// TIA Portal project "P11_2" (V20)

(* hardware
DEVICE "HMI_1"  KTP700 Basic PN
   slot 0: "HMI_1"  KTP700 Basic PN  6AV2 123-2GB03-0AX0  17.0.0.0
   slot 1: "HMI_RT_1"  KTP700 Basic PN  6AV2 123-2GB03-0AX0  17.0.0.0
   slot 5: "HMI_1.IE_CP_1"  PROFINET Interface  17.0.0.0
      slot 1: "PROFINET Interface_1"  PROFINET Interface
         slot 1: "Port_1"  Port
DEVICE "S7-1200 station_1"  S7-1200 Station
   slot 0: "Rack_0"  S7-1200 Rack  Rack  V1.0
   slot 1: "PLC_1"  CPU 1214C DC/DC/DC  6ES7 214-1AG40-0XB0  V4.7
*)

// ===== PLC "PLC_1"  CPU 1214C DC/DC/DC =====

VAR_GLOBAL   // PLC tag table "Default tag table"
   "Inicio" AT %M0.2 : Bool;
   "Marca 1" AT %M0.1 : Bool;
   "Marca0" AT %M0.0 : Bool;
   "Reset" AT %M0.4 : Bool;
   "SalidaControl" AT %M0.3 : Bool;
   "Tiempo_out_ms" AT %MD200 : Time;
   "Tiempo_out_seg" AT %MD66 : Real;
   "Tiempo_in" AT %MD150 : DInt;
   "Tiempo_in_ms" AT %MD184 : DInt;
   "Salida led" AT %M0.5 : Bool;
   "Regla3_1" AT %M26.0 : LReal;
   "Salida_barra" AT %M34.0 : LReal;
   "Tag_1" AT %Q0.0 : Bool;
   "Verde" AT %M2.0 : Bool;
   "Amarillo" AT %M2.1 : Bool;
   "Rojo" AT %M2.2 : Bool;
   "reset_rojo" AT %M2.3 : Bool;
   "reset_sem" AT %M2.4 : Bool;
   "cont_verde" AT %MD100 : Time;
   "cont_ama" AT %MD104 : Time;
   "cont_rojo" AT %MD108 : Time;
   "Tag_2" AT %MD12 : DInt;
   "T_restante" AT %MD16 : DInt;
   "Tag_3" AT %MD20 : DInt;
   "Tag_4" AT %MD24 : DInt;
   "Tag_5" AT %M26.0 : Bool;
   "Alarma1" AT %MW42 : Word;
   "bitalarma1" AT %M43.0 : Bool;
   "Alarma2" AT %MW44 : Word;
   "bitAlarma2" AT %M45.0 : Bool;
   "Alarma3" AT %MW46 : Word;
   "bitalarma3" AT %M47.0 : Bool;
END_VAR

// folder: System blocks/Program resources

DATA_BLOCK "IEC_Timer_0_DB"   // DB1
{ S7_Optimized_Access := 'TRUE' }
AUTHOR : Simatic
FAMILY : IEC
NAME : IEC_TMR
VERSION : 1.0
// stored: InstanceOfName IEC_TIMER
"IEC_TIMER"
BEGIN
END_DATA_BLOCK

DATA_BLOCK "IEC_Timer_0_DB_1"   // DB2
{ S7_Optimized_Access := 'TRUE' }
AUTHOR : Simatic
FAMILY : IEC
NAME : IEC_TMR
VERSION : 1.0
// stored: InstanceOfName IEC_TIMER
"IEC_TIMER"
BEGIN
END_DATA_BLOCK

DATA_BLOCK "IEC_Timer_0_DB_2"   // DB3
{ S7_Optimized_Access := 'TRUE' }
AUTHOR : Simatic
FAMILY : IEC
NAME : IEC_TMR
VERSION : 1.0
// stored: InstanceOfName IEC_TIMER
"IEC_TIMER"
BEGIN
END_DATA_BLOCK

DATA_BLOCK "IEC_Timer_0_DB_3"   // DB4
{ S7_Optimized_Access := 'TRUE' }
AUTHOR : Simatic
FAMILY : IEC
NAME : IEC_TMR
VERSION : 1.0
// stored: InstanceOfName IEC_TIMER
"IEC_TIMER"
BEGIN
END_DATA_BLOCK

// folder: (top level)

ORGANIZATION_BLOCK "Main"   // OB1, LAD, ProgramCycle
TITLE = "Main Program Sweep (Cycle)"
{ S7_Optimized_Access := 'TRUE' }
VERSION : 0.1
   VAR_INPUT
      Initial_Call : Bool;   // Initial call of this OB
      Remanence : Bool;   // =True, if remanent data are available
   END_VAR
BEGIN

REGION Network 1
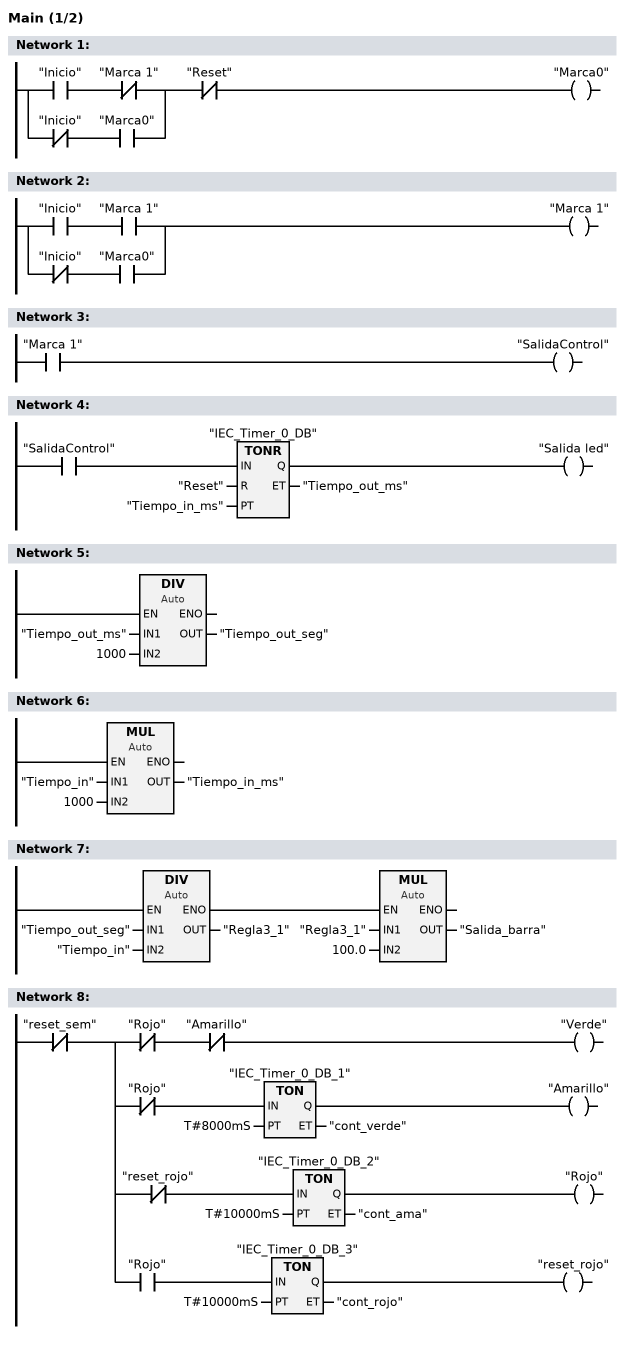
   RUNG wire#powerrail
      Contact( "Inicio" )
      I_Contact( "Marca 1" )
      wire#w1
      I_Contact( "Reset" )
      Coil( "Marca0" )
   END_RUNG
   RUNG wire#powerrail
      I_Contact( "Inicio" )
      Contact( "Marca0" )
   END_RUNG wire#w1
   // the same network as SCL:
   "Marca0" := (("Inicio" AND NOT "Marca 1") OR (NOT "Inicio" AND "Marca0")) AND NOT "Reset";
END_REGION

REGION Network 2
   RUNG wire#powerrail
      Contact( "Inicio" )
      Contact( "Marca 1" )
      wire#w1
      Coil( "Marca 1" )
   END_RUNG
   RUNG wire#powerrail
      I_Contact( "Inicio" )
      Contact( "Marca0" )
   END_RUNG wire#w1
   // the same network as SCL:
   "Marca 1" := ("Inicio" AND "Marca 1") OR (NOT "Inicio" AND "Marca0");
END_REGION

REGION Network 3
   RUNG wire#powerrail
      Contact( "Marca 1" )
      Coil( "SalidaControl" )
   END_RUNG
   // the same network as SCL:
   "SalidaControl" := "Marca 1";
END_REGION

REGION Network 4
   "IEC_Timer_0_DB".TONR(IN := "SalidaControl", R := "Reset", PT := "Tiempo_in_ms", ET => "Tiempo_out_ms");
   "Salida led" := "IEC_Timer_0_DB".Q;
END_REGION

REGION Network 5
   RUNG wire#powerrail
      Div(in1 := "Tiempo_out_ms", in2 := 1000, out => "Tiempo_out_seg")
   END_RUNG
   // the same network as SCL:
   "Tiempo_out_seg" := "Tiempo_out_ms" / 1000;
END_REGION

REGION Network 6
   RUNG wire#powerrail
      Mul(in1 := "Tiempo_in", in2 := 1000, out => "Tiempo_in_ms")
   END_RUNG
   // the same network as SCL:
   "Tiempo_in_ms" := "Tiempo_in" * 1000;
END_REGION

REGION Network 7
   RUNG wire#powerrail
      Div(in1 := "Tiempo_out_seg", in2 := "Tiempo_in", out => "Regla3_1")
      Mul(in1 := "Regla3_1", in2 := 100.0, out => "Salida_barra")
   END_RUNG
   // the same network as SCL:
   "Regla3_1" := "Tiempo_out_seg" / "Tiempo_in";
   "Salida_barra" := "Regla3_1" * 100.0;
END_REGION

REGION Network 8
   "Verde" := NOT "reset_sem" AND NOT "Rojo" AND NOT "Amarillo";
   "IEC_Timer_0_DB_1".TON(IN := NOT "reset_sem" AND NOT "Rojo", PT := T#8000mS, ET => "cont_verde");
   "Amarillo" := "IEC_Timer_0_DB_1".Q;
   "IEC_Timer_0_DB_2".TON(IN := NOT "reset_sem" AND NOT "reset_rojo", PT := T#10000mS, ET => "cont_ama");
   "Rojo" := "IEC_Timer_0_DB_2".Q;
   "IEC_Timer_0_DB_3".TON(IN := NOT "reset_sem" AND "Rojo", PT := T#10000mS, ET => "cont_rojo");
   "reset_rojo" := "IEC_Timer_0_DB_3".Q;
END_REGION

REGION Network 9
   // T restante verde
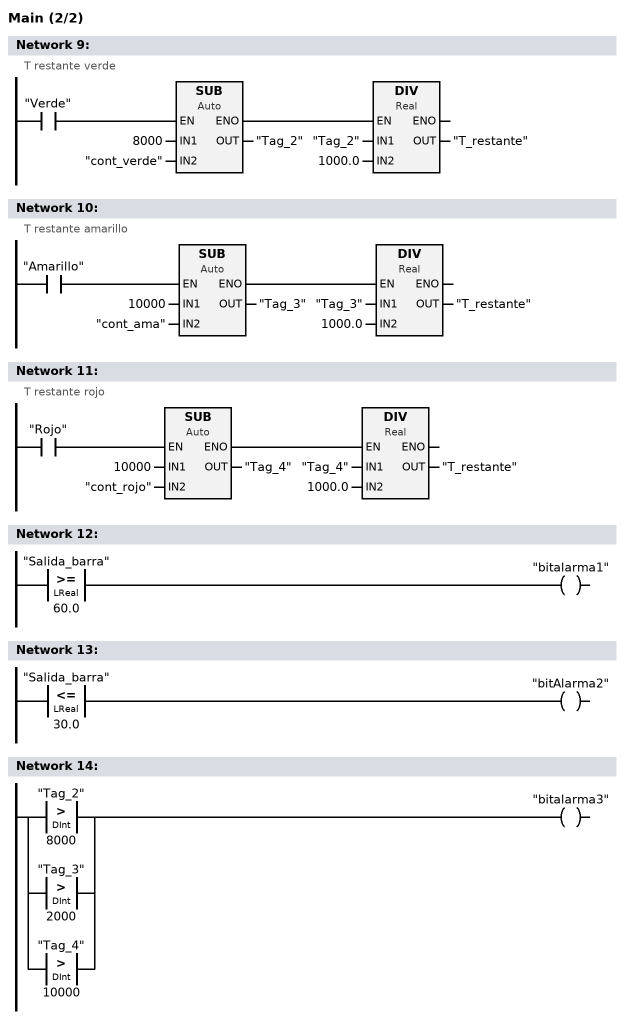
   RUNG wire#powerrail
      Contact( "Verde" )
      Sub(in1 := 8000, in2 := "cont_verde", out => "Tag_2")
      { S7_Templates := "SrcType := Real" } Div(in1 := "Tag_2", in2 := 1000.0, out => "T_restante")
   END_RUNG
   // the same network as SCL:
   IF "Verde" THEN
       "Tag_2" := 8000 - "cont_verde";
       "T_restante" := "Tag_2" / 1000.0;
   END_IF;
END_REGION

REGION Network 10
   // T restante amarillo
   RUNG wire#powerrail
      Contact( "Amarillo" )
      Sub(in1 := 10000, in2 := "cont_ama", out => "Tag_3")
      { S7_Templates := "SrcType := Real" } Div(in1 := "Tag_3", in2 := 1000.0, out => "T_restante")
   END_RUNG
   // the same network as SCL:
   IF "Amarillo" THEN
       "Tag_3" := 10000 - "cont_ama";
       "T_restante" := "Tag_3" / 1000.0;
   END_IF;
END_REGION

REGION Network 11
   // T restante rojo
   RUNG wire#powerrail
      Contact( "Rojo" )
      Sub(in1 := 10000, in2 := "cont_rojo", out => "Tag_4")
      { S7_Templates := "SrcType := Real" } Div(in1 := "Tag_4", in2 := 1000.0, out => "T_restante")
   END_RUNG
   // the same network as SCL:
   IF "Rojo" THEN
       "Tag_4" := 10000 - "cont_rojo";
       "T_restante" := "Tag_4" / 1000.0;
   END_IF;
END_REGION

REGION Network 12
   RUNG wire#powerrail
      { S7_Templates := "SrcType := LReal" } GE_Contact(in1 := "Salida_barra", in2 := 60.0)
      Coil( "bitalarma1" )
   END_RUNG
   // the same network as SCL:
   "bitalarma1" := "Salida_barra" >= 60.0;
END_REGION

REGION Network 13
   RUNG wire#powerrail
      { S7_Templates := "SrcType := LReal" } LE_Contact(in1 := "Salida_barra", in2 := 30.0)
      Coil( "bitAlarma2" )
   END_RUNG
   // the same network as SCL:
   "bitAlarma2" := "Salida_barra" <= 30.0;
END_REGION

REGION Network 14
   RUNG wire#powerrail
      { S7_Templates := "SrcType := DInt" } GT_Contact(in1 := "Tag_2", in2 := 8000)
      wire#w1
      Coil( "bitalarma3" )
   END_RUNG
   RUNG wire#powerrail
      { S7_Templates := "SrcType := DInt" } GT_Contact(in1 := "Tag_3", in2 := 2000)
   END_RUNG wire#w1
   RUNG wire#powerrail
      { S7_Templates := "SrcType := DInt" } GT_Contact(in1 := "Tag_4", in2 := 10000)
   END_RUNG wire#w1
   // the same network as SCL:
   "bitalarma3" := ("Tag_2" > 8000) OR ("Tag_3" > 2000) OR ("Tag_4" > 10000);
END_REGION
END_ORGANIZATION_BLOCK

(* ===== HMI "HMI_RT_1" =====
system functions are stored by id; their names below are inferred from use
connection "HMI_Connection_1": ETHERNET, SMART_S7_1200_OMS

HMI tags "Default tag table"
   "Tag_ScreenNumber" : UInt, internal
   "Inicio" : Bool = PLC Inicio AT %M0.2, 1 s
   "Reset" : Bool = PLC Reset AT %M0.4, 1 s
   "Tiempo_in" : DInt = PLC Tiempo_in AT %MD150, 1 s
   "Tiempo_out_seg" : Real = PLC Tiempo_out_seg AT %MD66, 1 s
   "Salida_barra" : LReal = PLC Salida_barra AT %M34.0, 1 s
   "Salida led" : Bool = PLC "Salida led" AT %M0.5, 1 s
   "Rojo" : Bool = PLC Rojo AT %M2.2, 1 s
   "Amarillo" : Bool = PLC Amarillo AT %M2.1, 1 s
   "Verde" : Bool = PLC Verde AT %M2.0, 1 s
   "T_restante" : DInt = PLC T_restante AT %MD16, 1 s
   "reset_sem" : Bool = PLC reset_sem AT %M2.4, 1 s
   "Alarma1" : Word = PLC Alarma1 AT %MW42, 1 s
   "Alarma2" : Word = PLC Alarma2 AT %MW44, 1 s
   "Alarma3" : Word = PLC Alarma3 AT %MW46, 1 s

discrete alarms
   1: 'Ha sobrepasado el 60%', class Errors, trigger "Alarma1" bit 0
   2: 'El nivel es menor al 30%', class Warnings, trigger "Alarma2" bit 0
   3: 'Tiempo establecido para cada estado no cumplido', class Acknowledgement, trigger "Alarma3" bit 0

text list "list_verde": 1 'AVANCE'; 0 ''

text list "list_rojo": 1 '¡ALTO!'; 0 ''

text list "list_ama": 1 'PRECAUCIÓN'; 0 ''

Template "Template_1" 800x480
   Button "Exit" at 714,429 size 71x50; TextOff 'Exit'; PictureOff "ExitRuntime_KTP700_Basic_PN_TR"; PictureOn "ExitRuntime_KTP700_Basic_PN_TR"
      on Release: StopRuntime(0)
   Button "Template_Button" at 614,429 size 71x50; TextOff 'Text'
   Button "Template_Button_1" at 514,429 size 71x50; TextOff 'Text'
   Button "Template_Button_2" at 414,429 size 71x50; TextOff 'Text'
   Button "Template_Button_3" at 314,429 size 71x50; TextOff 'Text'
   Button "Template_Button_4" at 214,429 size 71x50; TextOff 'Text'
   Button "Template_Button_5" at 114,429 size 71x50; TextOff 'Text'
   Button "Start screen" at 14,429 size 71x50; TextOff 'Start screen'; PictureOff "NavigateHome_KTP700_Basic_PN_TR"; PictureOn "NavigateHome_KTP700_Basic_PN_TR"
      on Release: ActivateScreen("Root screen", 0)
   SymbolicIOField "Symbolic_IO_Field_Screen" at 93,9 size 600x33; TextOff '0'; TextOn '1'; TextList "TextList_ScreenNames"
      ProcessValue <- "Tag_ScreenNumber"
      on Change: ActivateScreenByNumber("Tag_ScreenNumber", 0)
   DateTimeField "HmiScreenItemData" at 695,25 size 105x25
   DateTimeField "HmiScreenItemData_1" at 695,0 size 105x25
   GraphicView "Logo" at 0,0 size 91x51; Picture "Logo of HMI_1"

screen "Root screen" 800x480, template "Template_1"
   on GenerateScreen: SetTag("Tag_ScreenNumber", 1)
   Button "Button_1" at 633,377 size 145x32; TextOff 'Reset'
      on Press: SetBit("reset_sem")
      on Release: ResetBit("reset_sem")
   IOField "I/O field_1" at 455,160 size 79x39; FormatPattern 99; Unit s
      ProcessValue <- "T_restante"
   TextField "Text field_1" at 423,132 size 140x23; Text 'Tiempo restante'
   Circle "Circle_1" at 285,124 size 48x48
      Appearance <- "Rojo"
   Circle "Circle_2" at 284,199 size 48x48
      Appearance <- "Amarillo"
   Circle "Circle_3" at 283,267 size 48x48
      Appearance <- "Verde"
   SymbolicIOField "Symbolic I/O field_1" at 426,299 size 137x32; TextOff '0'; TextOn '1'; TextList "list_verde"
      ProcessValue <- "Verde"
   SymbolicIOField "Symbolic I/O field_2" at 426,264 size 136x32; TextOff '0'; TextOn '1'; TextList "list_ama"
      ProcessValue <- "Amarillo"
   SymbolicIOField "Symbolic I/O field_3" at 426,229 size 135x32; TextOff '0'; TextOn '1'; TextList "list_rojo"
      ProcessValue <- "Rojo"
   Button "FB_ArrowRight_Square" at 36,60 size 50x50; TextOff 'Text'; PictureOff "FB_ArrowRight_Square_Released_256c"; PictureOn "FB_ArrowRight_Square_Pressed_256c"
      on Press: ActivateScreen("tanque", 0)

screen "tanque" 800x480
   Bar "Bar_1" at 113,70 size 92x283; MinimumValue 0; MaximumValue 100
      ProcessValue <- "Salida_barra"
   TextField "Text field_1" at 249,149 size 143x23; Text 'Límite de tiempo'
   TextField "Text field_2" at 477,148 size 174x23; Text 'Tiempo Transcurrido'
   Button "Button_1" at 266,246 size 126x32; TextOff 'Inicio/Pausa'
      on Press: SetBit("Inicio")
      on Release: ResetBit("Inicio")
   Button "Button_2" at 477,246 size 128x32; TextOff 'Reset'
      on Press: SetBit("Reset")
      on Release: ResetBit("Reset")
   IOField "I/O field_1" at 267,177 size 96x32; FormatPattern 999; Unit  seg
      ProcessValue <- "Tiempo_in"
   IOField "I/O field_2" at 509,178 size 96x32; FormatPattern 999; Unit  seg
      ProcessValue <- "Tiempo_out_seg"
   Circle "Circle_1" at 416,246 size 34x34
      Appearance <- "Salida led"
   Button "FB_Home_Square" at 35,28 size 50x50; TextOff 'Text'; PictureOff "FB_Home_Square_Released_256c"; PictureOn "FB_Home_Square_Pressed_256c"
      on Press: ActivateScreen("Root screen", 0)
*)